(* IEC 61131-3 sources: eCockpitGit/test_project/src/%F%00 Library/%F%Common Functions/%F%Dynamic Array/%POU%FB_DynamicArray/%F%Internal, 2 files *)

(* ---- %METH%compare.st ---- *)
//Internal function to compare two elements correctly
// |**Version**|**Author**| **Date** |**Changes**
// | 1         | NSN      | 03-03-22 | Creation
METHOD PRIVATE compare : BOOL
VAR_INPUT
	elementInt		:POINTER TO BYTE;	//Internal element to compare
	elementExt		:POINTER TO BYTE;	//External element to compare
	elementExtSize	:WORD;				//Size of external element
END_VAR
VAR
	i				:WORD;
END_VAR
(*%!%__DELIMITER__%!%*)
IF S_strings OR elementExtSize = S_elementSize THEN
	//If first byte in element and first byte in array position are the same
	IF elementExt^ = elementInt^ THEN
		compare		:=		TRUE;
		IF S_elementSize > 1 THEN
			IF S_strings THEN
				//String array will account for zero termination
				FOR i := 0 TO S_elementSize - 1 DO
					IF elementExt[i] <> elementInt[i] THEN
						compare		:=		FALSE;
						EXIT;
					ELSIF elementExt[i] = 0 THEN
						IF elementInt[i] = 0 THEN
							EXIT;
						ELSE
							compare		:=		FALSE;
							EXIT;
						END_IF
					END_IF
				END_FOR
			ELSE
				//Normal type check entire element
				FOR i := 0 TO S_elementSize - 1 DO
					IF elementExt[i] <> elementInt[i] THEN
						compare		:=		FALSE;
						EXIT;
					END_IF
				END_FOR
			END_IF
		END_IF
	END_IF
END_IF

(* ---- %METH%FB_init.st ---- *)
//Reinitialization is not supported, so only set values once;
// |**Version**|**Author**| **Date** |**Changes**
// | 1         | NSN      | 03-03-22 | Creation
METHOD FB_Init: BOOL
VAR_INPUT
    bInitRetains		:BOOL; 		//TRUE: the retain variables are initialized (reset warm / reset cold)
    bInCopyCode			:BOOL;  	//TRUE: the instance will be copied to the copy code afterward (online change)
	pArray				:REFERENCE TO POINTER TO ARRAY[0..99] OF BYTE;	//Pointer to array pointer
	wIncrement			:WORD;		//How many element sizes are allocated when array size is increased
	wElementSize		:WORD;		//Size of individual element in array
	wMaxSize			:WORD;		//Max size allowed for array, 0 means no max
	xStringArray		:BOOL;		//Set true if the array contains only strings, as they should be compared with zero termination
	xMap				:BOOL;		//Set true for mapped mode, where duplicate elements cannot
END_VAR
(*%!%__DELIMITER__%!%*)
IF S_array = 0 THEN
	S_array				:=		ADR(pArray);
	S_increment			:=		wIncrement;
	S_elementSize		:=		wElementSize;
	IF wMaxSize = 0 THEN
		S_maxSize		:=		65535;
	ELSE
		S_maxSize		:=		wMaxSize;
	END_IF
	S_strings			:=		xStringArray;
	S_map				:=		xMap;
END_IF
